# EPICS substitutions: iocTops/_99Beers/db/user.substitutions
# Example substitutions file

file "db/dbExample1.db" {
    { user = "ktn98257" }
}
